// TIA Portal project "Ex7-Watertank_V16" (V16)
// The watertank project

(* hardware
DEVICE "S7-1200 station_1"  S7-1200 Station
   slot 0: "Rack_0"  S7-1200 Rack  Rack  V1.0
   slot 1: "PLC_1"  CPU 1215C DC/DC/Rly  6ES7 215-1HG40-0XB0  V4.2
*)

// ===== PLC "PLC_1"  CPU 1215C DC/DC/Rly =====

VAR_GLOBAL   // PLC tag table "Default tag table"
   "System_Byte" AT %MB254 : Byte;
   "FirstScan" AT %M254.0 : Bool;
   "DiagStatusUpdate" AT %M254.1 : Bool;
   "AlwaysTRUE" AT %M254.2 : Bool;
   "AlwaysFALSE" AT %M254.3 : Bool;
   "Clock_Byte" AT %MB255 : Byte;
   "Clock_10Hz" AT %M255.0 : Bool;
   "Clock_5Hz" AT %M255.1 : Bool;
   "Clock_2.5Hz" AT %M255.2 : Bool;
   "Clock_2Hz" AT %M255.3 : Bool;
   "Clock_1.25Hz" AT %M255.4 : Bool;
   "Clock_1Hz" AT %M255.5 : Bool;
   "Clock_0.625Hz" AT %M255.6 : Bool;
   "Clock_0.5Hz" AT %M255.7 : Bool;
END_VAR

VAR_GLOBAL   // PLC tag table "Tag table_FIO"
   "oT1_VlvIn_U21" AT %QD100 : Real;   // Inlet valve
   "oT1_VlvOut_U22" AT %QD104 : Real;   // Outlet valve
   "iT1_SenLev_S21" AT %ID100 : Real;   // Level sensor tank T1
   "iT1_SenFlow_S22" AT %ID104 : Real;   // Flow sensor outlet tank T1
END_VAR

VAR_GLOBAL   // PLC tag table "Tag table_ASTIO"
   "iCC_BtnStop_S1" AT %I0.0 : Bool;   // Stop button
   "iCC_BtnStart_S3" AT %I0.2 : Bool;   // Start button
   "iCC_BtnReset_S5" AT %I0.4 : Bool;   // Reset button
   "oCC_LmpStart_H1" AT %Q0.0 : Bool;   // Lamp start
   "oCC_LmpErr_H3" AT %Q0.2 : Bool;   // Lamp error
   "iCC_PotLev_R1" AT %IW64 : Int;   // Potentiometer level setpoint
END_VAR

VAR_GLOBAL   // PLC tag table "Tag table_Flags"
   "mA001" AT %M0.0 : Bool;   // Alarm high level exceeded
   "mA001_016" AT %MW0 : Word;   // Reserverd for alarms A001 to A016
   "mT1_SenLev_mm" AT %MD2 : Real;   // Level tank 1 [mm]
   "mT1_FlowLev_ls" AT %MD6 : Real;   // Flow outlet tank 1 l/s]
   "mT1_VlvIn_perc" AT %MD10 : Real;   // Inlet valve [%]
   "mT1_VlvOut_perc" AT %MD14 : Real;   // Outlet valve [%]
   "mGenStarted" AT %M30.0 : Bool;   // Installation started
   "mT1_Fill" AT %M30.1 : Bool;   // Fill tank T1
   "mT1_Temp" AT %MD18 : Real;   // Temporary value
   "mT1_SP" AT %MD22 : Real;   // Level setpoint [mm]
END_VAR

// folder: System blocks/Program resources

DATA_BLOCK "ID_TON_T1_Lev"   // DB1
{ S7_Optimized_Access := 'TRUE' }
AUTHOR : Simatic
FAMILY : IEC
NAME : IEC_TMR
VERSION : 1.0
// stored: InstanceOfName IEC_TIMER
"IEC_TIMER"
BEGIN
END_DATA_BLOCK

// folder: (top level)

FUNCTION "FC_CC" : Void   // FC1, FBD
TITLE = Control cabinet
{ S7_Optimized_Access := 'TRUE' }
VERSION : 0.1
BEGIN

REGION Network 1: Start-stop control circuit
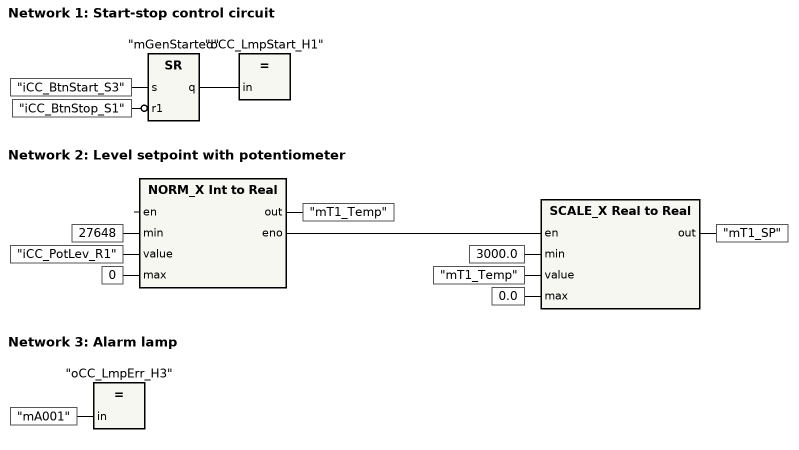
   IF "iCC_BtnStart_S3" THEN
       "mGenStarted" := TRUE;   // SR flip-flop
   END_IF;
   IF NOT "iCC_BtnStop_S1" THEN "mGenStarted" := FALSE; END_IF;
   "oCC_LmpStart_H1" := "mGenStarted";
END_REGION

REGION Network 2: Level setpoint with potentiometer
   // The max. setpoint value is equal to the height of the tank
   "mT1_Temp" := NORM_X(MIN := 27648, VALUE := "iCC_PotLev_R1", MAX := 0);
   "mT1_SP" := SCALE_X(MIN := 3000.0, VALUE := "mT1_Temp", MAX := 0.0);
END_REGION

REGION Network 3: Alarm lamp
   "oCC_LmpErr_H3" := "mA001";
END_REGION
END_FUNCTION

FUNCTION "FC_T1" : Void   // FC2, FBD
TITLE = Tank 1
{ S7_Optimized_Access := 'TRUE' }
VERSION : 0.1
BEGIN

REGION Network 1: AD Conversion level sensor
   // Remark: Factory IO range = 0.0 .. 10.0 (REAL) instead of 0 ... 27648 (INT)
   // 3 m = 3000 mm
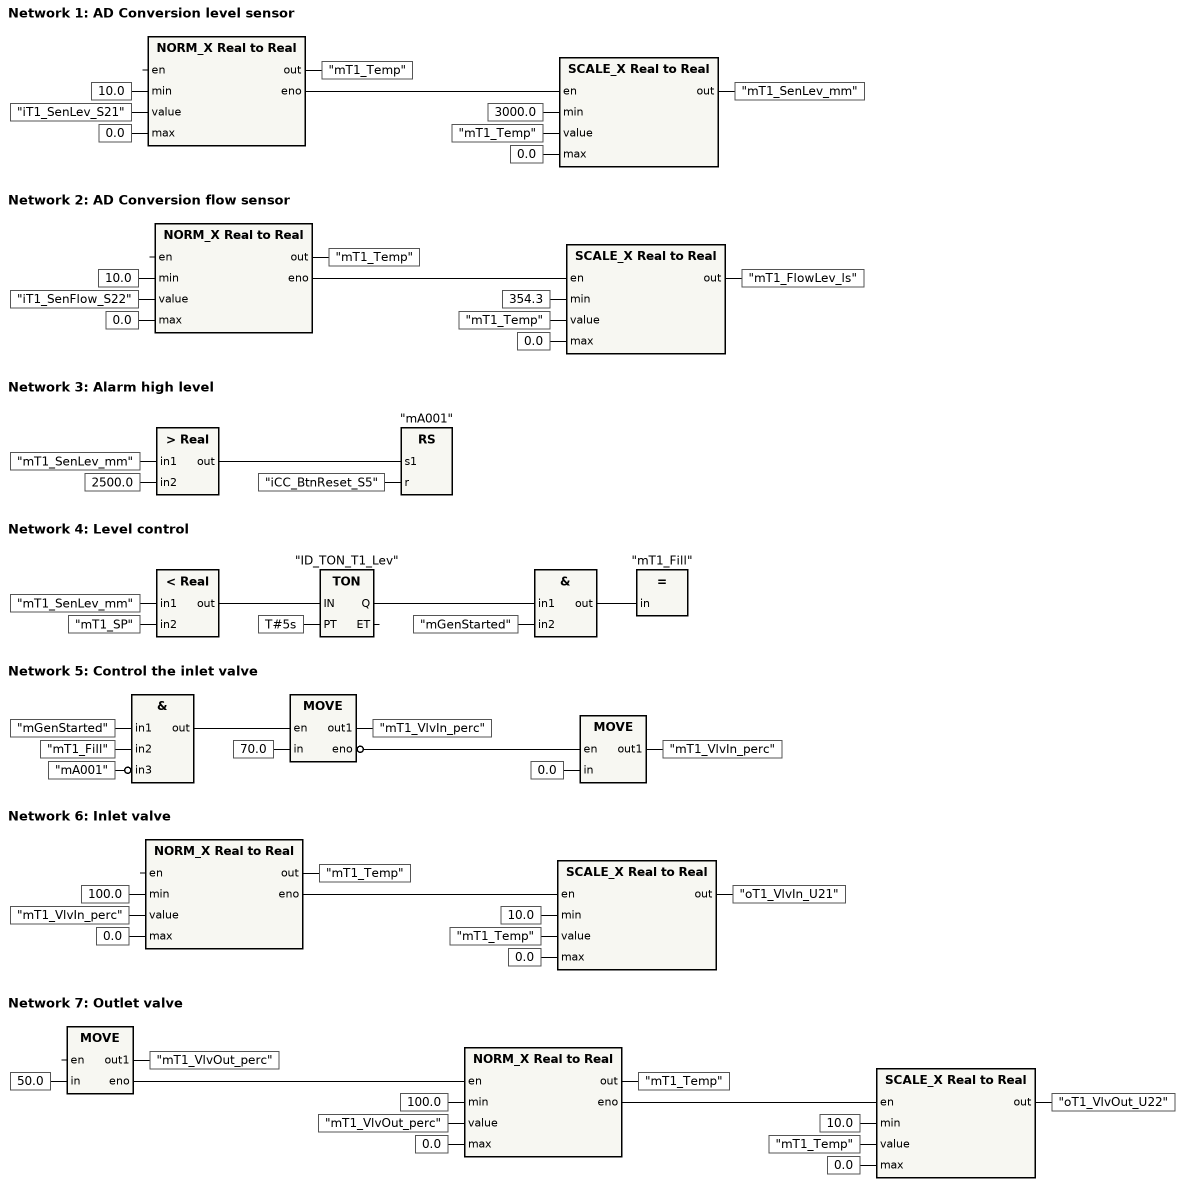
   "mT1_Temp" := NORM_X(MIN := 10.0, VALUE := "iT1_SenLev_S21", MAX := 0.0);
   "mT1_SenLev_mm" := SCALE_X(MIN := 3000.0, VALUE := "mT1_Temp", MAX := 0.0);
END_REGION

REGION Network 2: AD Conversion flow sensor
   // Remark: Factory IO range = 0.0 .. 10.0 (REAL) instead of 0 ... 27648 (INT)
   // 0,3543 m³/s = 354,3 l/s
   "mT1_Temp" := NORM_X(MIN := 10.0, VALUE := "iT1_SenFlow_S22", MAX := 0.0);
   "mT1_FlowLev_ls" := SCALE_X(MIN := 354.3, VALUE := "mT1_Temp", MAX := 0.0);
END_REGION

REGION Network 3: Alarm high level
   IF "iCC_BtnReset_S5" THEN
       "mA001" := FALSE;   // RS flip-flop
   END_IF;
   IF "mT1_SenLev_mm" > 2500.0 THEN "mA001" := TRUE; END_IF;
END_REGION

REGION Network 4: Level control
   "ID_TON_T1_Lev".TON(IN := "mT1_SenLev_mm" < "mT1_SP", PT := T#5s);
   "mT1_Fill" := "ID_TON_T1_Lev".Q AND "mGenStarted";
END_REGION

REGION Network 5: Control the inlet valve
   IF "mGenStarted" AND "mT1_Fill" AND NOT "mA001" THEN "mT1_VlvIn_perc" := 70.0; END_IF;
   IF NOT ("mGenStarted" AND "mT1_Fill" AND NOT "mA001") THEN "mT1_VlvIn_perc" := 0.0; END_IF;
END_REGION

REGION Network 6: Inlet valve
   "mT1_Temp" := NORM_X(MIN := 100.0, VALUE := "mT1_VlvIn_perc", MAX := 0.0);
   "oT1_VlvIn_U21" := SCALE_X(MIN := 10.0, VALUE := "mT1_Temp", MAX := 0.0);
END_REGION

REGION Network 7: Outlet valve
   // Outlet valve always for 50% open (even we the installation is stopped)
   "mT1_VlvOut_perc" := 50.0;
   "mT1_Temp" := NORM_X(MIN := 100.0, VALUE := "mT1_VlvOut_perc", MAX := 0.0);
   "oT1_VlvOut_U22" := SCALE_X(MIN := 10.0, VALUE := "mT1_Temp", MAX := 0.0);
END_REGION
END_FUNCTION

ORGANIZATION_BLOCK "Main"   // OB1, FBD, ProgramCycle
TITLE = "Main Program Sweep (Cycle)"
{ S7_Optimized_Access := 'TRUE' }
VERSION : 0.1
   VAR_INPUT
      Initial_Call : Bool;   // Initial call of this OB
      Remanence : Bool;   // =True, if remanent data are available
   END_VAR
BEGIN

REGION Network 1: Control cabinet
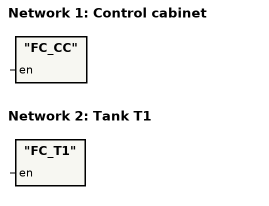
   "FC_CC"();
END_REGION

REGION Network 2: Tank T1
   "FC_T1"();
END_REGION
END_ORGANIZATION_BLOCK